// TIA Portal V19 export
DATA_BLOCK "Areas_ITF"   // DB3
// stored: Access Published, MemoryReserve 100
   VAR
      A01 : "ITF_A01";
      A02 : "ITF_A02";
      A03 : "ITF_A03";
      A04 : "ITF_A04";
      AG : "ITF_AG";
      Prod { S7_SetPoint := 'True'} : "ITF_ProductionMng";
   END_VAR
BEGIN
END_DATA_BLOCK
